{attribute 'GeneratedUsingTerminal: EJ3318-0000-0017'}
{attribute addProperty BoxType "EJ3318-0000-0017"}
{attribute addProperty Id "StatusAT %I*Status_68C33E995ValueAT %I*INT2"}
{attribute addProperty CRC "2507538081"}
{attribute addProperty Size "7"}
TYPE TC_Channel_9575FEA1 :
STRUCT
	{attribute addProperty Name "Status"}
	Status AT %I* : Status_68C33E99;
	{attribute addProperty Name "Value"}
	Value AT %I* : INT;
END_STRUCT
END_TYPE

(* stored: Version 1.2.0.0, ProductVersion 3.1.4024.9
   DUT TC_Channel_9575FEA1: Id {fe16ded0-8ead-4f90-9762-b6d9fd040439} *)
